// TIA Portal V17 export
// export: Created 2024-08-07T21:44:13.3582013Z, ExportSetting WithDefaults, DisplayName Totally Integrated Automation Portal, DisplayVersion V17 Update 7, DisplayName TIA Portal Openness, DisplayVersion V17 Update 7, DisplayName TIA Portal Version Control Interface, DisplayVersion V17, DisplayName SINAMICS Startdrive Advanced, DisplayVersion V17 SP2, DisplayName SINAMICS Startdrive G110M, G120, G120C, G120D, G120P, G115D, DisplayVersion V17 SP2, DisplayName SINAMICS Startdrive G130, G150, S120, S150, SINAMICS MV, S210, DisplayVersion V17 SP2, DisplayName STEP 7 Professional, DisplayVersion V17 Update 7, DisplayName STEP 7 Safety, DisplayVersion V17 Update 6, DisplayName WinCC Advanced / Unified PC, DisplayVersion V17 Update 7
VAR_GLOBAL   // PLC tag table "Data Costant"
END_VAR
VAR_GLOBAL CONSTANT   // user constants
   MaxCreateNFP : Int := 10;   // Number of max creating NFP²s
   MaxDataReading : Int := 25;   // Number of max data reading
   MaxRoundNumber : Int := 1;   // Number of Rounds
   NumberOfmessages : Int := 6;   // Number of messages from IJCore
   MaxStageStep : Int := 25;   // Number of Max Step Step
   MaxInitStep : Int := 2;   // Number of Max Init Step
   MaxRobot : Int := 3;   // Number of Max Robot
   MaxReader : Int := 5;   // Number of Max Reader
   MaxSolenoid : Int := 48;   // Number of Max Solenoid
   NotUsed : Int := 0;
   MasterNFP : Int := 2;
   SecondaryNFP : Int := 3;
   Component : Int := 4;
   STA : Int := 1;
   PFC : Int := 2;
   TRW : Int := 3;
   TRI : Int := 4;
   TRR : Int := 5;
   CMA : Int := 7;
   TMA : Int := 8;
   CNF : Int := 9;
   TRC : Int := 10;
   TRS : Int := 6;
   TRB : Int := 11;
END_VAR
